//Assert
AssertEquals_INT(E_ProfidriveGSM_State.S1_SwitchingOnInhibited, fbFSM.eState, 'eState: AssertEquals not returning expected value');

TEST_FINISHED();


TEST('Transition S51>S52');

//Arrange
fbFSM.bPowerOn := TRUE;
fbFSM.eState := E_ProfidriveGSM_State.S51_RampStop;

fbFSM.bStandstill					:= FALSE;
fbFSM.stSTW1.b0_On 				:= FALSE;
fbFSM.stSTW1.b1_CoastStop 		:= TRUE;
fbFSM.stSTW1.b2_QuickStop 		:= FALSE;
fbFSM.stSTW1.b3_EnableOperation 	:= TRUE;

//Act
fbFSM();

//Assert
AssertEquals_INT(E_ProfidriveGSM_State.S52_QuickStop, fbFSM.eState, 'eState: AssertEquals not returning expected value');

TEST_FINISHED();


TEST('Transition S51>S2 Case_1');

//Arrange
fbFSM.bPowerOn := TRUE;
fbFSM.eState := E_ProfidriveGSM_State.S51_RampStop;

fbFSM.bStandstill					:= FALSE;
fbFSM.stSTW1.b0_On 				:= FALSE;
fbFSM.stSTW1.b1_CoastStop 		:= TRUE;
fbFSM.stSTW1.b2_QuickStop 		:= TRUE;
fbFSM.stSTW1.b3_EnableOperation 	:= FALSE;

//Act
fbFSM();

//Assert
AssertEquals_INT(E_ProfidriveGSM_State.S2_ReadyForSwitchingOn, fbFSM.eState, 'eState: AssertEquals not returning expected value');

TEST_FINISHED();


TEST('Transition S51>S2 Case_2');

//Arrange
fbFSM.bPowerOn := TRUE;
fbFSM.eState := E_ProfidriveGSM_State.S51_RampStop;

fbFSM.bStandstill					:= TRUE;
fbFSM.stSTW1.b0_On 				:= FALSE;
fbFSM.stSTW1.b1_CoastStop 		:= TRUE;
fbFSM.stSTW1.b2_QuickStop 		:= TRUE;
fbFSM.stSTW1.b3_EnableOperation 	:= TRUE;

//Act
fbFSM();

//Assert
AssertEquals_INT(E_ProfidriveGSM_State.S2_ReadyForSwitchingOn, fbFSM.eState, 'eState: AssertEquals not returning expected value');

TEST_FINISHED();


TEST('Transition S51>S4');

//Arrange
fbFSM.bPowerOn := TRUE;
fbFSM.eState := E_ProfidriveGSM_State.S51_RampStop;

fbFSM.bStandstill					:= FALSE;
fbFSM.stSTW1.b0_On 				:= TRUE;
fbFSM.stSTW1.b1_CoastStop 		:= TRUE;
fbFSM.stSTW1.b2_QuickStop 		:= TRUE;
fbFSM.stSTW1.b3_EnableOperation 	:= TRUE;

//Act
fbFSM();

//Assert
AssertEquals_INT(E_ProfidriveGSM_State.S4_Operation, fbFSM.eState, 'eState: AssertEquals not returning expected value');

TEST_FINISHED();
END_METHOD

METHOD TestTransitions_S52 : BOOL
VAR
	fbFSM 				: FB_ProfidriveGSM;
	stStatusExpected	: ST_ProfiidriveGSM_ZSW1;
	nStatusExpected 	: WORD;
END_VAR
TEST('Transition S52 Still');

//Arrange
fbFSM.bPowerOn := TRUE;
fbFSM.eState := E_ProfidriveGSM_State.S52_QuickStop;

fbFSM.bStandstill					:= FALSE;
fbFSM.stSTW1.b0_On 				:= FALSE;
fbFSM.stSTW1.b1_CoastStop 		:= TRUE;
fbFSM.stSTW1.b2_QuickStop 		:= FALSE;
fbFSM.stSTW1.b3_EnableOperation 	:= TRUE;

//Act
fbFSM();

//Assert
AssertEquals_INT(E_ProfidriveGSM_State.S52_QuickStop, fbFSM.eState, 'eState: AssertEquals not returning expected value');

TEST_FINISHED();


TEST('Transition S51>S1 Case_1');

//Arrange
fbFSM.bPowerOn := TRUE;
fbFSM.eState := E_ProfidriveGSM_State.S52_QuickStop;

fbFSM.bStandstill					:= FALSE;
fbFSM.stSTW1.b0_On 				:= FALSE;
fbFSM.stSTW1.b1_CoastStop 		:= FALSE;
fbFSM.stSTW1.b2_QuickStop 		:= FALSE;
fbFSM.stSTW1.b3_EnableOperation 	:= FALSE;

//Act
fbFSM();

//Assert
AssertEquals_INT(E_ProfidriveGSM_State.S1_SwitchingOnInhibited, fbFSM.eState, 'eState: AssertEquals not returning expected value');

TEST_FINISHED();


TEST('Transition S52>S1 Case_2');

//Arrange
fbFSM.bPowerOn := TRUE;
fbFSM.eState := E_ProfidriveGSM_State.S52_QuickStop;

fbFSM.bStandstill					:= FALSE;
fbFSM.stSTW1.b0_On 				:= FALSE;
fbFSM.stSTW1.b1_CoastStop 		:= TRUE;
fbFSM.stSTW1.b2_QuickStop 		:= FALSE;
fbFSM.stSTW1.b3_EnableOperation 	:= FALSE;

//Act
fbFSM();

//Assert
AssertEquals_INT(E_ProfidriveGSM_State.S1_SwitchingOnInhibited, fbFSM.eState, 'eState: AssertEquals not returning expected value');

TEST_FINISHED();

TEST('Transition S52>S1 Case_3');

//Arrange
fbFSM.bPowerOn := TRUE;
fbFSM.eState := E_ProfidriveGSM_State.S52_QuickStop;

fbFSM.bStandstill					:= TRUE;
fbFSM.stSTW1.b0_On 				:= FALSE;
fbFSM.stSTW1.b1_CoastStop 		:= TRUE;
fbFSM.stSTW1.b2_QuickStop 		:= FALSE;
fbFSM.stSTW1.b3_EnableOperation 	:= TRUE;

//Act
fbFSM();

//Assert
AssertEquals_INT(E_ProfidriveGSM_State.S1_SwitchingOnInhibited, fbFSM.eState, 'eState: AssertEquals not returning expected value');

TEST_FINISHED();
END_METHOD

END_FUNCTION_BLOCK

// Tests/Drives/FB_ProfidriveTelegram1_Test
FUNCTION_BLOCK FB_ProfidriveTelegram1_Test EXTENDS TcUnit.FB_TestSuite

Test_ProcessDataControl();
Test_ProcessDataStatus();

METHOD Test_ProcessDataControl : REFERENCE TO FB_Test
VAR
	fbDrive 					: FB_ProfidriveTelegram1;
	
	nExpectedSTW1 				: WORD;
	nExpectedNSOLL				: INT;
	nActualSTW1 				: WORD;
	nActualNSOLL				: INT;	
	
	aExpectedControlData 		: ARRAY[1..4] OF BYTE;
	aExpectedStatusData 		: ARRAY[1..4] OF BYTE;
END_VAR
TEST('Assign Process data Control');

//Arrange
nExpectedSTW1 := 16#A1B2;
nExpectedNSOLL 	:= UINT_TO_INT(16#C3D4);
F_Memcpy(ADR(aExpectedControlData), ADR(nExpectedSTW1), 2, FALSE);
F_Memcpy(ADR(aExpectedControlData) + 2, ADR(nExpectedNSOLL), 2, FALSE);
fbDrive.AssignProcessData(aExpectedControlData, aExpectedStatusData);

//Act
fbDrive.GetControlData();

//Assert
F_Memcpy(ADR(nActualSTW1), ADR(fbDrive.stControl), 2, FALSE);
F_Memcpy(ADR(nActualNSOLL), ADR(fbDrive.stControl) + 2, 2, FALSE);

AssertEquals(Expected := nExpectedSTW1,
             Actual := nActualSTW1,
             Message := 'nSTW1 is not correct');
	 
AssertEquals(Expected := nExpectedNSOLL,
             Actual := nActualNSOLL,
             Message := 'nNSOLL is not correct');	

TEST_FINISHED();


TEST('Assign Process data Control Swap');

//Arrange
nExpectedSTW1 := 16#C3F3;
nExpectedNSOLL 	:= UINT_TO_INT(16#C3F3);
F_Memcpy(ADR(aExpectedControlData), ADR(nExpectedSTW1), 2, TRUE);
F_Memcpy(ADR(aExpectedControlData) + 2, ADR(nExpectedNSOLL), 2, TRUE);

fbDrive.stConfig.bSwapProcessData := TRUE;
fbDrive.AssignProcessData(aExpectedControlData, aExpectedStatusData);

//Act
fbDrive.GetControlData();

//Assert
F_Memcpy(ADR(nActualSTW1), ADR(fbDrive.stControl), 2, FALSE);
F_Memcpy(ADR(nActualNSOLL), ADR(fbDrive.stControl) + 2, 2, FALSE);

AssertEquals(Expected := nExpectedSTW1,
             Actual := nActualSTW1,
             Message := 'nSTW1 is not correct');
	 
AssertEquals(Expected := nExpectedNSOLL,
             Actual := nActualNSOLL,
             Message := 'nNSOLL is not correct');	

TEST_FINISHED();
END_METHOD

METHOD Test_ProcessDataStatus : REFERENCE TO FB_Test
VAR
	fbDrive 					: FB_ProfidriveTelegram1;
	
	nExpectedZSW1 				: WORD;
	nExpectedNIST				: INT;	
	nActualZSW1 				: WORD;
	nActualNIST					: INT;	

	aExpectedControlData 		: ARRAY[1..4] OF BYTE;	
	aExpectedStatusData 		: ARRAY[1..4] OF BYTE;	
END_VAR
TEST('Assign Process data Status');

//Arrange
nExpectedZSW1 := 16#A1B2;
nExpectedNIST 	:= UINT_TO_INT(16#C3D4);
F_Memcpy(ADR(fbDrive.stStatus), ADR(nExpectedZSW1), 2, FALSE);
F_Memcpy(ADR(fbDrive.stStatus) + 2, ADR(nExpectedNIST), 2, FALSE);
fbDrive.AssignProcessData(aExpectedControlData, aExpectedStatusData);

//Act
fbDrive.SetStatusData();

//Assert
F_Memcpy(ADR(nActualZSW1), ADR(aExpectedStatusData), 2, FALSE);
F_Memcpy(ADR(nActualNIST), ADR(aExpectedStatusData) + 2, 2, FALSE);

AssertEquals(Expected := nExpectedZSW1,
             Actual := nActualZSW1,
             Message := 'nZSW1 is not correct');
	 
AssertEquals(Expected := nExpectedNIST,
             Actual := nActualNIST,
             Message := 'nNIST is not correct');	

TEST_FINISHED();


TEST('Assign Process data Status SWAP');

//Arrange
nExpectedZSW1 := 16#A1B2;
nExpectedNIST 	:= UINT_TO_INT(16#C3D4);
F_Memcpy(ADR(fbDrive.stStatus), ADR(nExpectedZSW1), 2, FALSE);
F_Memcpy(ADR(fbDrive.stStatus) + 2, ADR(nExpectedNIST), 2, FALSE);
fbDrive.AssignProcessData(aExpectedControlData, aExpectedStatusData);
fbDrive.stConfig.bSwapProcessData := TRUE;

//Act
fbDrive.SetStatusData();

//Assert
F_Memcpy(ADR(nActualZSW1), ADR(aExpectedStatusData), 2, TRUE);
F_Memcpy(ADR(nActualNIST), ADR(aExpectedStatusData) + 2, 2, TRUE);

AssertEquals(Expected := nExpectedZSW1,
             Actual := nActualZSW1,
             Message := 'nZSW1 is not correct');
	 
AssertEquals(Expected := nExpectedNIST,
             Actual := nActualNIST,
             Message := 'nNIST is not correct');	

TEST_FINISHED();
END_METHOD

END_FUNCTION_BLOCK

// Tests/PRG_TEST
PROGRAM PRG_TEST
VAR
	FB_ProfidriveGSM_Test : FB_ProfidriveGSM_Test;
	FB_ProfidriveTelegram1_Test : FB_ProfidriveTelegram1_Test;
END_VAR

TcUnit.RUN();

END_PROGRAM
